INTERFACE I_DigitalInput

PROPERTY isActive : bool
GET
END_GET
END_PROPERTY

PROPERTY isNotActive : bool
GET
END_GET
END_PROPERTY

END_INTERFACE

(* stored: Version 1.1.0.1, ProductVersion 3.1.4026.18
   Itf I_DigitalInput: Id {7822e320-9a93-4f41-9965-14007ab1f275}
   Property isActive: Id {968b9e9a-5732-4778-bcd2-1ae5f41cba56}
   Get Get: Id {158f3797-4945-444a-9141-fcc66aead7ac}
   Property isNotActive: Id {22fe28d0-669d-4a1f-9ad4-b6c5043fdef8}
   Get Get: Id {303b0784-ee8f-4ec3-8de2-b8071fcf7b1e} *)
